INTERFACE I_NotificationHandler EXTENDS __SYSTEM.IQueryInterface

METHOD OnNotificationReceived
VAR_INPUT
    NotificationId   : UDINT;
    NotificationName : T_MaxString;
    Args             : I_StreamReader;
END_VAR
END_METHOD

END_INTERFACE

(* stored: Version 1.1.0.1, ProductVersion 3.1.4024.6
   Itf I_NotificationHandler: Id {132ee55d-2226-43c5-82b5-622b17ca944c}
   Method OnNotificationReceived: Id {600e8039-a73b-451c-9206-c0585bf94fa7} *)
